// TIA Portal V17 export
// export: Created 2024-09-03T21:54:59.0184409Z, ExportSetting WithDefaults, DisplayName Totally Integrated Automation Portal, DisplayVersion V17 Update 7, DisplayName TIA Portal Openness, DisplayVersion V17 Update 7, DisplayName TIA Portal Version Control Interface, DisplayVersion V17, DisplayName SINAMICS Startdrive Advanced, DisplayVersion V17 SP2, DisplayName SINAMICS Startdrive G110M, G120, G120C, G120D, G120P, G115D, DisplayVersion V17 SP2, DisplayName SINAMICS Startdrive G130, G150, S120, S150, SINAMICS MV, S210, DisplayVersion V17 SP2, DisplayName STEP 7 Professional, DisplayVersion V17 Update 7, DisplayName STEP 7 Safety, DisplayVersion V17 Update 6, DisplayName WinCC Advanced / Unified PC, DisplayVersion V17 Update 7
FUNCTION_BLOCK "sq_manipulator"   // FB44, GRAPH
VERSION : 0.1
// stored: AcknowledgeErrorsRequired true, AutoNumber true, GraphVersion 6.0, InitialValuesAcquisition false, IsIECCheckEnabled false, LanguageInNetworks LAD, LockOperatingMode false, PermanentILProcessingInMANMode false, SetENOAutomatically false, SkipSteps false, UDAEnableTagReadback false, WithAlarmHandling true
   // inherited from GRAPH_BASE
   VAR
      OFF_SQ_BASE : Bool;
   END_VAR
   VAR_INPUT
      OFF_SQ { ExternalAccessible := 'False'; ExternalVisible := 'False'; ExternalWritable := 'False'} : Bool := false;   // Turn sequence off
      INIT_SQ { ExternalAccessible := 'False'; ExternalVisible := 'False'; ExternalWritable := 'False'} : Bool := false;   // Set sequence to initial state
      ACK_EF { ExternalAccessible := 'False'; ExternalVisible := 'False'; ExternalWritable := 'False'} : Bool := false;   // Acknowledge all errors and faults
      S_PREV { ExternalAccessible := 'False'; ExternalVisible := 'False'; ExternalWritable := 'False'} : Bool := false;   // Output previous step in parameter S_NO
      S_NEXT { ExternalAccessible := 'False'; ExternalVisible := 'False'; ExternalWritable := 'False'} : Bool := false;   // Indicate next step in parameter S_NO
      SW_AUTO { ExternalAccessible := 'False'; ExternalVisible := 'False'; ExternalWritable := 'False'} : Bool := false;   // Automatic mode
      SW_TAP { ExternalAccessible := 'False'; ExternalVisible := 'False'; ExternalWritable := 'False'} : Bool := false;   // Semiautomatic/switch with transition
      SW_TOP { ExternalAccessible := 'False'; ExternalVisible := 'False'; ExternalWritable := 'False'} : Bool := false;   // Semiautomatic/ignore transition
      SW_MAN { ExternalAccessible := 'False'; ExternalVisible := 'False'; ExternalWritable := 'False'} : Bool := false;   // Manual mode
      S_SEL { ExternalAccessible := 'False'; ExternalVisible := 'False'; ExternalWritable := 'False'} : Int := 0;   // Select step to be output to S_NO
      S_ON { ExternalAccessible := 'False'; ExternalVisible := 'False'; ExternalWritable := 'False'} : Bool := false;   // Activate step indicated in S_NO
      S_OFF { ExternalAccessible := 'False'; ExternalVisible := 'False'; ExternalWritable := 'False'} : Bool := false;   // Deactivate step indicated S_NO
      T_PUSH { ExternalAccessible := 'False'; ExternalVisible := 'False'; ExternalWritable := 'False'} : Bool := false;   // Enable transition to switch in semi automatic mode
   END_VAR
   VAR_OUTPUT
      S_NO { ExternalAccessible := 'False'; ExternalVisible := 'False'; ExternalWritable := 'False'} : Int := 0;   // Step number
      S_MORE { ExternalAccessible := 'False'; ExternalVisible := 'False'; ExternalWritable := 'False'} : Bool := false;   // More steps are available and can be shown in S_NO
      S_ACTIVE { ExternalAccessible := 'False'; ExternalVisible := 'False'; ExternalWritable := 'False'} : Bool := false;   // Step indicated in S_NO is active
      ERR_FLT { ExternalAccessible := 'False'; ExternalVisible := 'False'; ExternalWritable := 'False'} : Bool := false;   // Interlock or supervision group error
      AUTO_ON { ExternalAccessible := 'False'; ExternalVisible := 'False'; ExternalWritable := 'False'} : Bool := false;   // Automatic mode is active
      TAP_ON { ExternalAccessible := 'False'; ExternalVisible := 'False'; ExternalWritable := 'False'} : Bool := false;   // Semiautomatic mode/step with transition enabled
      TOP_ON { ExternalAccessible := 'False'; ExternalVisible := 'False'; ExternalWritable := 'False'} : Bool := false;   // Semiautomatic mode/ignore transition enabled
      MAN_ON { ExternalAccessible := 'False'; ExternalVisible := 'False'; ExternalWritable := 'False'} : Bool := false;   // Manual mode is active
   END_VAR
   VAR
      dummy : Bool;
      start : Bool;
      base : Bool;
      IEC_Timer_0_Instance { S7_SetPoint := 'True'} : TON_TIME;
      IEC_Timer_0_Instance_1 { S7_SetPoint := 'True'} : TON_TIME;
      IEC_Timer_0_Instance_2 { S7_SetPoint := 'True'} : TON_TIME;
   END_VAR
BEGIN
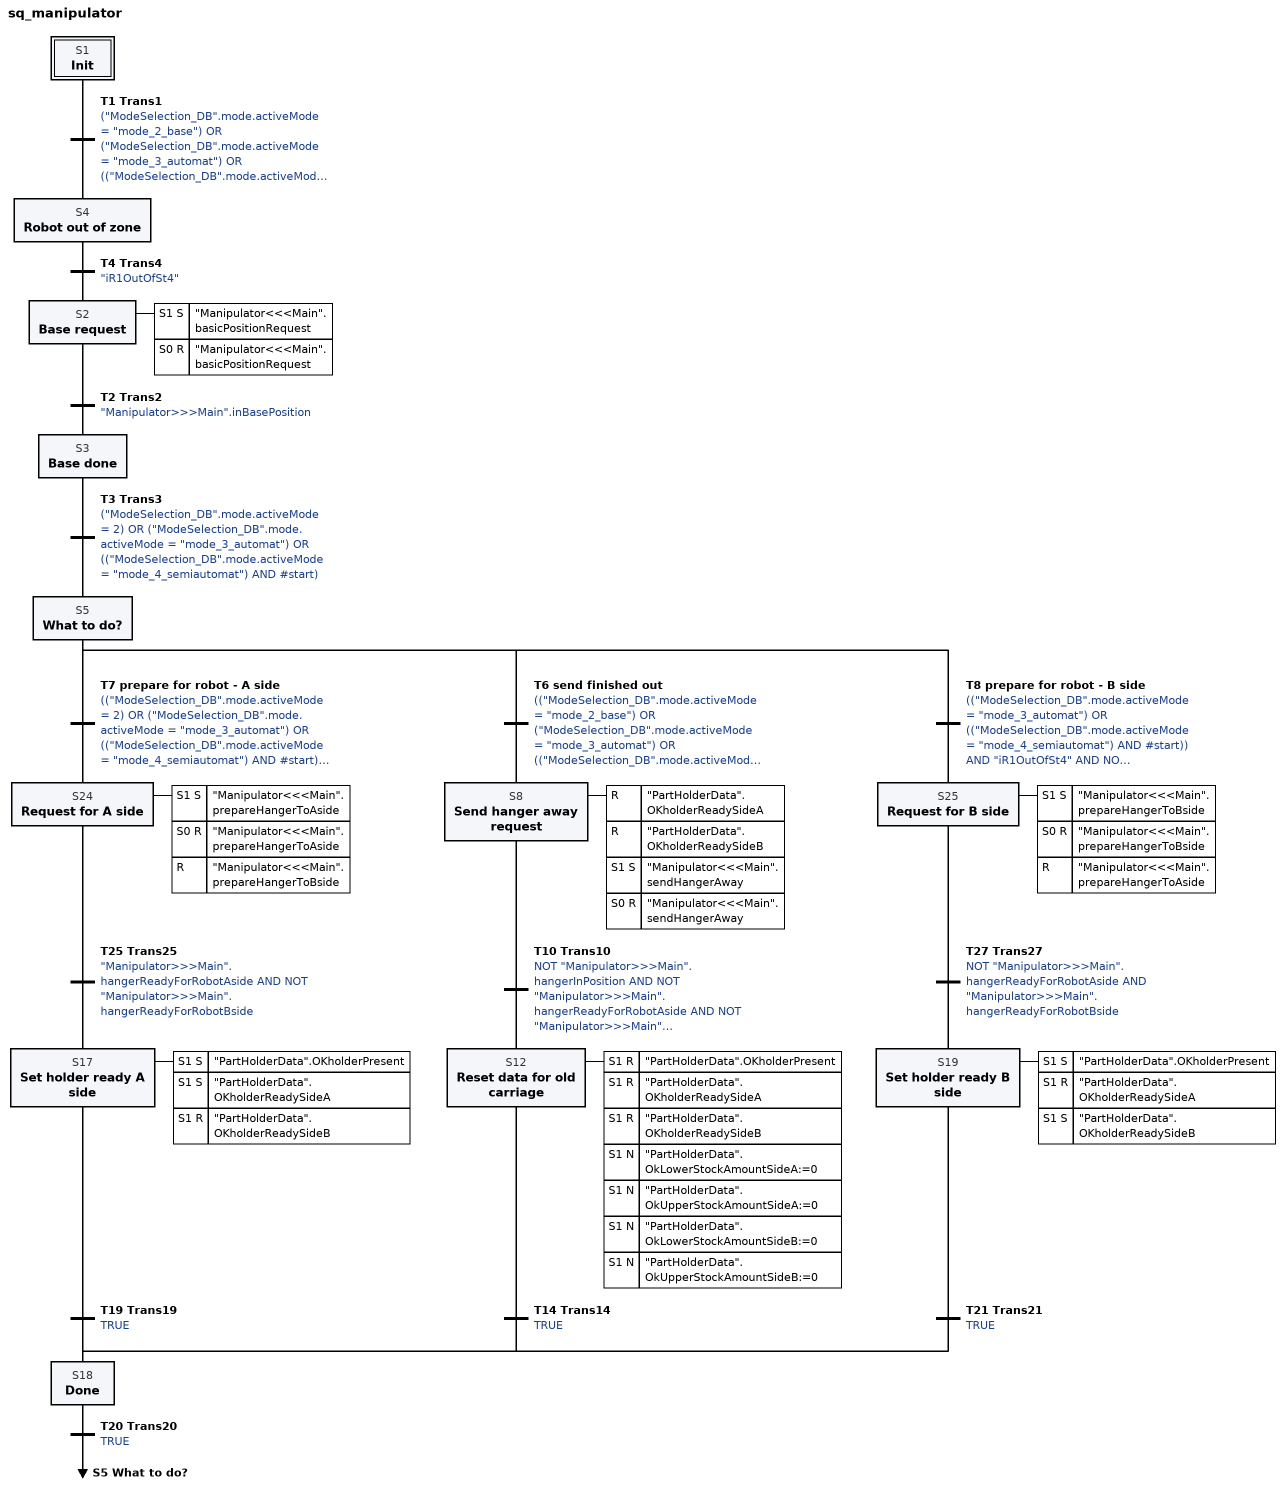
   // permanent pre-instructions
   NETWORK 1
   TITLE = base
      #base := #"Base done".X;

   // sequencer 1
   INITIAL_STEP Init:   // S1, max time T#10S, warning time T#7S
   END_STEP
   TRANSITION Trans1 FROM Init TO "Robot out of zone"   // T1
      := ("ModeSelection_DB".mode.activeMode = "mode_2_base") OR ("ModeSelection_DB".mode.activeMode = "mode_3_automat") OR (("ModeSelection_DB".mode.activeMode = "mode_4_semiautomat") AND #start);
   END_TRANSITION
   STEP "Base request":   // S2, max time T#10S, warning time T#7S
          S1  S    "Manipulator<<<Main".basicPositionRequest
          S0  R    "Manipulator<<<Main".basicPositionRequest
   END_STEP
   TRANSITION Trans2 FROM "Base request" TO "Base done"   // T2
      := "Manipulator>>>Main".inBasePosition;
   END_TRANSITION
   STEP "Base done":   // S3, max time T#10S, warning time T#7S
   END_STEP
   TRANSITION Trans3 FROM "Base done" TO "What to do?"   // T3
      := ("ModeSelection_DB".mode.activeMode = 2) OR ("ModeSelection_DB".mode.activeMode = "mode_3_automat") OR (("ModeSelection_DB".mode.activeMode = "mode_4_semiautomat") AND #start);
   END_TRANSITION
   STEP "Robot out of zone":   // S4, max time T#10S, warning time T#7S
      supervision V := (#"Robot out of zone".T > #"Robot out of zone".T_MAX) AND (T#0MS > #"Robot out of zone".T_MAX);
   END_STEP
   TRANSITION Trans4 FROM "Robot out of zone" TO "Base request"   // T4
      := "iR1OutOfSt4";
   END_TRANSITION
   STEP "What to do?":   // S5, max time T#10S, warning time T#7S
   END_STEP
   TRANSITION "prepare for robot - A side" FROM "What to do?" TO "Request for A side"   // T7
      := (("ModeSelection_DB".mode.activeMode = 2) OR ("ModeSelection_DB".mode.activeMode = "mode_3_automat") OR (("ModeSelection_DB".mode.activeMode = "mode_4_semiautomat") AND #start)) AND "iR1OutOfSt4" AND NOT "PartHolderData".OKholderReadySideA AND (("PartHolderData".OkLowerStockAmountSideA < "StationParameters".OKLowerStockSize) OR ("PartHolderData".OkUpperStockAmountSideA < "StationParameters".OKUpperStockSize));
   END_TRANSITION
   TRANSITION "send finished out" FROM "What to do?" TO "Send hanger away request"   // T6
      := (("ModeSelection_DB".mode.activeMode = "mode_2_base") OR ("ModeSelection_DB".mode.activeMode = "mode_3_automat") OR (("ModeSelection_DB".mode.activeMode = "mode_4_semiautomat") AND #start)) AND "iR1OutOfSt4" AND "PartHolderData".OKholderPresent AND ((("PartHolderData".OkLowerStockAmountSideA >= "StationParameters".OKLowerStockSize) AND ("PartHolderData".OkUpperStockAmountSideA >= "StationParameters".OKUpperStockSize) AND ("PartHolderData".OkLowerStockAmountSideB >= "StationParameters".OKLowerStockSize) AND ("PartHolderData".OkUpperStockAmountSideB >= "StationParameters".OKUpperStockSize)) OR "Manipulator<<<Main".reserve[0].%X0) AND NOT "sq_robot_"."Dropoff part to manipulator level1".X AND NOT "sq_robot_"."Dropoff part to manipulator level2".X;
   END_TRANSITION
   TRANSITION "prepare for robot - B side" FROM "What to do?" TO "Request for B side"   // T8
      := (("ModeSelection_DB".mode.activeMode = "mode_3_automat") OR (("ModeSelection_DB".mode.activeMode = "mode_4_semiautomat") AND #start)) AND "iR1OutOfSt4" AND NOT "PartHolderData".OKholderReadySideB AND (("PartHolderData".OkLowerStockAmountSideB < "StationParameters".OKLowerStockSize) OR ("PartHolderData".OkUpperStockAmountSideB < "StationParameters".OKUpperStockSize)) AND ("PartHolderData".OkLowerStockAmountSideA >= "StationParameters".OKLowerStockSize) AND ("PartHolderData".OkUpperStockAmountSideA >= "StationParameters".OKUpperStockSize);
   END_TRANSITION
   STEP "Request for B side":   // S25, max time T#30S, warning time T#7S
      supervision V := (#"Request for B side".T > #"Request for B side".T_MAX) AND (T#0MS > #"Request for B side".T_MAX);
          S1  S    "Manipulator<<<Main".prepareHangerToBside
          S0  R    "Manipulator<<<Main".prepareHangerToBside
              R    "Manipulator<<<Main".prepareHangerToAside
   END_STEP
   TRANSITION Trans27 FROM "Request for B side" TO "Set holder ready B side"   // T27
      := NOT "Manipulator>>>Main".hangerReadyForRobotAside AND "Manipulator>>>Main".hangerReadyForRobotBside;
   END_TRANSITION
   STEP "Set holder ready A side":   // S17, max time T#10S, warning time T#7S
          S1  S    "PartHolderData".OKholderPresent
          S1  S    "PartHolderData".OKholderReadySideA
          S1  R    "PartHolderData".OKholderReadySideB
   END_STEP
   TRANSITION Trans19 FROM "Set holder ready A side" TO Done   // T19
      := TRUE;
   END_TRANSITION
   STEP Done:   // S18, max time T#10S, warning time T#7S
   END_STEP
   TRANSITION Trans20 FROM Done TO "What to do?"   // T20, jump
      := TRUE;
   END_TRANSITION
   STEP "Send hanger away request":   // S8, max time T#10S, warning time T#7S
              R    "PartHolderData".OKholderReadySideA
              R    "PartHolderData".OKholderReadySideB
          S1  S    "Manipulator<<<Main".sendHangerAway
          S0  R    "Manipulator<<<Main".sendHangerAway
   END_STEP
   TRANSITION Trans10 FROM "Send hanger away request" TO "Reset data for old carriage"   // T10
      := NOT "Manipulator>>>Main".hangerInPosition AND NOT "Manipulator>>>Main".hangerReadyForRobotAside AND NOT "Manipulator>>>Main".hangerReadyForRobotBside;
   END_TRANSITION
   STEP "Set holder ready B side":   // S19, max time T#10S, warning time T#7S
          S1  S    "PartHolderData".OKholderPresent
          S1  R    "PartHolderData".OKholderReadySideA
          S1  S    "PartHolderData".OKholderReadySideB
   END_STEP
   TRANSITION Trans21 FROM "Set holder ready B side" TO Done   // T21
      := TRUE;
   END_TRANSITION
   STEP "Reset data for old carriage":   // S12, max time T#10S, warning time T#7S
          S1  R    "PartHolderData".OKholderPresent
          S1  R    "PartHolderData".OKholderReadySideA
          S1  R    "PartHolderData".OKholderReadySideB
          S1  N    "PartHolderData".OkLowerStockAmountSideA:=0
          S1  N    "PartHolderData".OkUpperStockAmountSideA:=0
          S1  N    "PartHolderData".OkLowerStockAmountSideB:=0
          S1  N    "PartHolderData".OkUpperStockAmountSideB:=0
   END_STEP
   TRANSITION Trans14 FROM "Reset data for old carriage" TO Done   // T14
      := TRUE;
   END_TRANSITION
   STEP "Request for A side":   // S24, max time T#30S, warning time T#7S
      supervision V := (#"Request for A side".T > #"Request for A side".T_MAX) AND (T#0MS > #"Request for A side".T_MAX);
          S1  S    "Manipulator<<<Main".prepareHangerToAside
          S0  R    "Manipulator<<<Main".prepareHangerToAside
              R    "Manipulator<<<Main".prepareHangerToBside
   END_STEP
   TRANSITION Trans25 FROM "Request for A side" TO "Set holder ready A side"   // T25
      := "Manipulator>>>Main".hangerReadyForRobotAside AND NOT "Manipulator>>>Main".hangerReadyForRobotBside;
   END_TRANSITION
END_FUNCTION_BLOCK
